METHOD GroupBuild : E_PROGRESS
VAR_INPUT
  Execute     : BOOL;
END_VAR
VAR_INST
  _nErrorId   : UDINT;
  _eJobReslt,
  _eState     : E_PROGRESS;
END_VAR
//-----------------------------------------------------------------------------
IF NOT Execute 
THEN 
	_eState                       := E_PROGRESS.PROGRESS_INIT; 
END_IF 
//-----------------------------------------------------------------------------
IF NOT Check() 
THEN 
	GroupBuild                    := E_PROGRESS.PROGRESS_ERROR; 
	RETURN; 
END_IF
//-----------------------------------------------------------------------------
//-----------------------------------------------------------------------------
CASE _eState
OF
  E_PROGRESS.PROGRESS_INIT:
    IF Execute
    THEN
      _nErrorId                 := 0;

      IF (_GroupInfo.AxisCount <> 0)
      THEN
        _nErrorId               := 9999;
        _eState                 := E_PROGRESS.PROGRESS_ERROR;
      ELSE
        _eState                 := E_PROGRESS.PROGRESS_BUSY;
        _eJobReslt              := _GroupItf.AddAll(FALSE);
      END_IF
    END_IF
END_CASE
//---------------------------------------------------------------------------
//---------------------------------------------------------------------------
CASE _eState
OF
  E_PROGRESS.PROGRESS_BUSY:
    _eJobReslt                  := _GroupItf.AddAll(TRUE);

    IF (_eJobReslt = E_PROGRESS.PROGRESS_ERROR)
    THEN
      _eState                   := E_PROGRESS.PROGRESS_ERROR;

      _nErrorId                 := _GroupInfo.GroupErrorId;
      _eJobReslt                := _GroupItf.AddAll(FALSE);

    ELSIF (_eJobReslt = E_PROGRESS.PROGRESS_DONE)
    THEN
      _eState                   := E_PROGRESS.PROGRESS_DONE;
      _eJobReslt                := _GroupItf.AddAll(FALSE);
    END_IF
END_CASE
//-----------------------------------------------------------------------------
//-----------------------------------------------------------------------------

GroupBuild                      := _eState;
END_METHOD

METHOD GroupClear : E_PROGRESS
VAR_INPUT
  Execute     : BOOL;
END_VAR
VAR_INST
  _nErrorId   : UDINT;
  _eJobReslt,
  _eState     : E_PROGRESS;
END_VAR
//-----------------------------------------------------------------------------
IF NOT Execute 
THEN 
	_eState                       := E_PROGRESS.PROGRESS_INIT; 
END_IF 
//-----------------------------------------------------------------------------
IF NOT Check() 
THEN 
	GroupClear                    := E_PROGRESS.PROGRESS_ERROR; 
	RETURN; 
END_IF
//-----------------------------------------------------------------------------
//-----------------------------------------------------------------------------
CASE _eState
OF
  E_PROGRESS.PROGRESS_INIT:
    IF Execute
    THEN
      _nErrorId                 := 0;
      _eJobReslt                := _GroupItf.McHaltAll(FALSE);
      _eState                   := E_PROGRESS.PROGRESS_BUSY;
    END_IF
  //---------------------------------------------------------------------------
  //---------------------------------------------------------------------------
  E_PROGRESS.PROGRESS_BUSY:
    _eJobReslt                  := _GroupItf.McHaltAll(TRUE);

    IF (_eJobReslt = E_PROGRESS.PROGRESS_ERROR)
    THEN
      _eState                   := E_PROGRESS.PROGRESS_ERROR;
      _nErrorId                 := _GroupInfo.GroupErrorId;
      _eJobReslt                := _GroupItf.McHaltAll(FALSE);

    ELSIF (_eJobReslt = E_PROGRESS.PROGRESS_DONE)
    THEN
      _eState                   := E_PROGRESS.PROGRESS_PREPARE;
      _eJobReslt                := _GroupItf.McResetAll(FALSE);
      _eJobReslt                := _GroupItf.McHaltAll(FALSE);
    END_IF
  //---------------------------------------------------------------------------
  //---------------------------------------------------------------------------
  E_PROGRESS.PROGRESS_PREPARE:
    _eJobReslt                  := _GroupItf.McResetAll(TRUE);

    IF (_eJobReslt = E_PROGRESS.PROGRESS_ERROR)
    THEN
      _eState                   := E_PROGRESS.PROGRESS_ERROR;
      _nErrorId                 := _GroupInfo.GroupErrorId;
      _eJobReslt                := _GroupItf.McResetAll(FALSE);

    ELSIF (_eJobReslt = E_PROGRESS.PROGRESS_DONE)
    THEN
      _eState                   := E_PROGRESS.PROGRESS_STARTUP;
      _eJobReslt                := _GroupItf.McResetAll(FALSE);
      _eJobReslt                := _GroupItf.RemoveAll(FALSE);
    END_IF
  //---------------------------------------------------------------------------
  //---------------------------------------------------------------------------
  E_PROGRESS.PROGRESS_STARTUP:
    _eJobReslt                  := _GroupItf.RemoveAll(TRUE);

    IF (_eJobReslt = E_PROGRESS.PROGRESS_ERROR)
    THEN
      _eState                   := E_PROGRESS.PROGRESS_ERROR;
      _nErrorId                 := _GroupInfo.GroupErrorId;
      _eJobReslt                := _GroupItf.RemoveAll(FALSE);

    ELSIF (_eJobReslt = E_PROGRESS.PROGRESS_DONE)
    THEN
      _eState                   := E_PROGRESS.PROGRESS_CHECK;
      _eJobReslt                := _GroupItf.RemoveAll(FALSE);
      _eJobReslt                := _GroupItf.Disable(FALSE);
    END_IF
  //---------------------------------------------------------------------------
  //---------------------------------------------------------------------------
  E_PROGRESS.PROGRESS_CHECK:
    _eJobReslt                  := _GroupItf.Disable(TRUE);

    IF (_eJobReslt = E_PROGRESS.PROGRESS_ERROR)
    THEN
      _eState                   := E_PROGRESS.PROGRESS_ERROR;
      _nErrorId                 := _GroupInfo.GroupErrorId;
      _eJobReslt                := _GroupItf.Disable(FALSE);

    ELSIF (_eJobReslt = E_PROGRESS.PROGRESS_DONE)
    THEN
      _eState                   := E_PROGRESS.PROGRESS_OCCUPIED;
      _eJobReslt                := _GroupItf.Disable(FALSE);
      _eJobReslt                := _GroupItf.Reset(FALSE);
    END_IF
  //---------------------------------------------------------------------------
  //---------------------------------------------------------------------------
  E_PROGRESS.PROGRESS_OCCUPIED:
    _eJobReslt                 := _GroupItf.Reset(TRUE);

    IF (_eJobReslt = E_PROGRESS.PROGRESS_ERROR)
    THEN
      _eState                   := E_PROGRESS.PROGRESS_ERROR;
      _nErrorId                 := _GroupInfo.GroupErrorId;
      _eJobReslt                := _GroupItf.Reset(FALSE);

    ELSIF (_eJobReslt = E_PROGRESS.PROGRESS_DONE)
    THEN
      _eState                   := E_PROGRESS.PROGRESS_WORKING;
      _eJobReslt                := _GroupItf.Reset(FALSE);
    END_IF
END_CASE
//-----------------------------------------------------------------------------
//-----------------------------------------------------------------------------
CASE _eState
OF
  E_PROGRESS.PROGRESS_WORKING:
    IF (_GroupInfo.GroupDisabled) AND NOT
       (_GroupInfo.GroupError)
    THEN
      _eState                   := E_PROGRESS.PROGRESS_DONE;
    ELSE
      IF (_GroupInfo.GroupErrorStop) OR
         (_GroupInfo.GroupError)
      THEN
        _eState                 := E_PROGRESS.PROGRESS_ERROR;
      END_IF
    END_IF
END_CASE
//-----------------------------------------------------------------------------
//-----------------------------------------------------------------------------

GroupClear                      := _eState;
END_METHOD

METHOD GroupEnable : E_PROGRESS
VAR_INPUT
  Execute     : BOOL;
END_VAR
VAR_INST
  _nErrorId   : UDINT;
  _eJobReslt,
  _eState     : E_PROGRESS;
END_VAR
//-----------------------------------------------------------------------------
IF NOT Execute 
THEN 
	_eState                       := E_PROGRESS.PROGRESS_INIT; 
END_IF 
//-----------------------------------------------------------------------------
IF NOT Check() 
THEN 
	GroupEnable                   := E_PROGRESS.PROGRESS_ERROR; 
	RETURN; 
END_IF
//-----------------------------------------------------------------------------
//-----------------------------------------------------------------------------
CASE _eState
OF
  E_PROGRESS.PROGRESS_INIT:
    IF Execute
    THEN
      _nErrorId                 := 0;

      IF NOT (_GroupInfo.AxisCount <> 0)
      THEN
        _nErrorId               := 9999;
        _eState                 := E_PROGRESS.PROGRESS_ERROR;
      ELSE
        _eState                 := E_PROGRESS.PROGRESS_BUSY;
        _eJobReslt              := _GroupItf.Enable(FALSE);
      END_IF
    END_IF
END_CASE
//---------------------------------------------------------------------------
//---------------------------------------------------------------------------
CASE _eState
OF
  E_PROGRESS.PROGRESS_BUSY:
    _eJobReslt                  := _GroupItf.Enable(TRUE);

    IF (_eJobReslt = E_PROGRESS.PROGRESS_ERROR)
    THEN
      _eState                   := E_PROGRESS.PROGRESS_ERROR;

      _nErrorId                 := _GroupInfo.GroupErrorId;
      _eJobReslt                := _GroupItf.Enable(FALSE);

    ELSIF (_eJobReslt = E_PROGRESS.PROGRESS_DONE)
    THEN
      _eState                   := E_PROGRESS.PROGRESS_CHECK;
      _eJobReslt                := _GroupItf.Enable(FALSE);
    END_IF
END_CASE
//-----------------------------------------------------------------------------
//-----------------------------------------------------------------------------
CASE _eState
OF
  E_PROGRESS.PROGRESS_CHECK:
    IF (_GroupInfo.GroupStandby) OR
       (_GroupInfo.GroupMoving)  OR
       (_GroupInfo.GroupNotReady)
    THEN
      _eState                   := E_PROGRESS.PROGRESS_DONE;
    ELSE
      IF (_GroupInfo.GroupErrorStop) OR
         (_GroupInfo.GroupError)
      THEN
        _eState                 := E_PROGRESS.PROGRESS_ERROR;
      END_IF
    END_IF
END_CASE
//-----------------------------------------------------------------------------
//-----------------------------------------------------------------------------
GroupEnable                     := _eState;
END_METHOD

PROPERTY GroupInfo : REFERENCE TO ST_GROUP_INFO
SET
_GroupInfo REF= GroupInfo;
END_SET
END_PROPERTY

PROPERTY GroupItf : I_XtsTransport_CaGroup
SET
_GroupItf := GroupItf;
END_SET
END_PROPERTY

METHOD MoverDisableAll : e_progress
VAR_INPUT
  Execute     : BOOL;
END_VAR
VAR_INST
  _nMover     : UINT;
  _nErrorId   : UDINT;
  _eRslt,
  _eState     : E_PROGRESS;
END_VAR
//-----------------------------------------------------------------------------
IF NOT Execute 
THEN 
	_eState                       := E_PROGRESS.PROGRESS_INIT; 
END_IF 
//-----------------------------------------------------------------------------
IF NOT Check() 
THEN 
	MoverDisableAll               := E_PROGRESS.PROGRESS_ERROR; 
	RETURN; 
END_IF
//-----------------------------------------------------------------------------
//-----------------------------------------------------------------------------
CASE _eState
OF
  E_PROGRESS.PROGRESS_INIT:
    IF Execute
    THEN
      _nErrorId                 := 0;
      _nMover                   := 1;

      _eState                   := E_PROGRESS.PROGRESS_BUSY;
    END_IF
END_CASE
//-----------------------------------------------------------------------------
//-----------------------------------------------------------------------------
CASE _eState
OF
  E_PROGRESS.PROGRESS_BUSY:
    _eState                     := E_PROGRESS.PROGRESS_PREPARE;
    _eRslt                      := _MoverItf[_nMover].Disable(FALSE);
END_CASE
//-----------------------------------------------------------------------------
//-----------------------------------------------------------------------------
CASE _eState
OF
  E_PROGRESS.PROGRESS_PREPARE:
    _eRslt                      := _MoverItf[_nMover].Disable(TRUE);

    IF (_eRslt = E_PROGRESS.PROGRESS_ERROR)
    THEN
      _eState                   := E_PROGRESS.PROGRESS_ERROR;
      _nErrorId                 := _MoverInfo[_nMover].nErrorId; 

    ELSIF (_eRslt = E_PROGRESS.PROGRESS_DONE)
    THEN
      _eState                   := E_PROGRESS.PROGRESS_STARTUP;
    END_IF
END_CASE
//-----------------------------------------------------------------------------
//-----------------------------------------------------------------------------
CASE _eState
OF
  E_PROGRESS.PROGRESS_STARTUP:
    _eState                     := E_PROGRESS.PROGRESS_CHECK;
    _eRslt                      := _MoverItf[_nMover].Disable(FALSE);
END_CASE
//-----------------------------------------------------------------------------
//-----------------------------------------------------------------------------
CASE _eState
OF
  E_PROGRESS.PROGRESS_CHECK:
    IF (_nMover > MAX_MOVER-1)
    THEN
      _eState                   := E_PROGRESS.PROGRESS_DONE;
    ELSE
      _nMover                   := _nMover + 1;
      _eState                   := E_PROGRESS.PROGRESS_BUSY;
    END_IF
END_CASE
//-----------------------------------------------------------------------------
//-----------------------------------------------------------------------------

MoverDisableAll                 := _eState;
END_METHOD

METHOD MoverEnableAll : e_progress
VAR_INPUT
  Execute     : BOOL;
END_VAR
VAR_INST
  _nMover     : UINT;
  _nErrorId   : UDINT;
  _eRslt,
  _eState     : E_PROGRESS;
END_VAR
//-----------------------------------------------------------------------------
IF NOT Execute 
THEN 
	_eState                       := E_PROGRESS.PROGRESS_INIT; 
END_IF 
//-----------------------------------------------------------------------------
IF NOT Check() 
THEN 
	MoverEnableAll                := E_PROGRESS.PROGRESS_ERROR; 
	RETURN; 
END_IF
//-----------------------------------------------------------------------------
//-----------------------------------------------------------------------------
CASE _eState
OF
  E_PROGRESS.PROGRESS_INIT:
    IF Execute
    THEN
      _nErrorId                 := 0;
      _nMover                   := 1;

      _eState                   := E_PROGRESS.PROGRESS_BUSY;
    END_IF
END_CASE
//-----------------------------------------------------------------------------
//-----------------------------------------------------------------------------
CASE _eState
OF
  E_PROGRESS.PROGRESS_BUSY:
    _eState                     := E_PROGRESS.PROGRESS_PREPARE;
    _eRslt                      := _MoverItf[_nMover].Enable(FALSE);
END_CASE
//-----------------------------------------------------------------------------
//-----------------------------------------------------------------------------
CASE _eState
OF
  E_PROGRESS.PROGRESS_PREPARE:
    _eRslt                      := _MoverItf[_nMover].Enable(TRUE);

    IF (_eRslt = E_PROGRESS.PROGRESS_ERROR)
    THEN
      _eState                   := E_PROGRESS.PROGRESS_ERROR;
      _nErrorId                 := _MoverInfo[_nMover].nErrorId; 

    ELSIF (_eRslt = E_PROGRESS.PROGRESS_DONE)
    THEN
      _eState                   := E_PROGRESS.PROGRESS_STARTUP;
    END_IF
END_CASE
//-----------------------------------------------------------------------------
//-----------------------------------------------------------------------------
CASE _eState
OF
  E_PROGRESS.PROGRESS_STARTUP:
    _eState                     := E_PROGRESS.PROGRESS_CHECK;
    _eRslt                      := _MoverItf[_nMover].Enable(FALSE);
END_CASE
//-----------------------------------------------------------------------------
//-----------------------------------------------------------------------------
CASE _eState
OF
  E_PROGRESS.PROGRESS_CHECK:
    IF (_nMover > MAX_MOVER-1)
    THEN
      _eState                   := E_PROGRESS.PROGRESS_DONE;
    ELSE
      _nMover                   := _nMover + 1;
      _eState                   := E_PROGRESS.PROGRESS_BUSY;
    END_IF
END_CASE
//-----------------------------------------------------------------------------
//-----------------------------------------------------------------------------

MoverEnableAll                  := _eState;
END_METHOD

PROPERTY MoverInfo : REFERENCE TO ARRAY[1..MAX_MOVER] OF ST_MOVER_INFO
SET
_MoverInfo REF= MoverInfo;
END_SET
END_PROPERTY

PROPERTY MoverItf : reference TO ARRAY[1..MAX_MOVER] OF I_XtsTransport_Mover
SET
_MoverItf REF= MoverItf;
END_SET
END_PROPERTY

PROPERTY StartStationIndex : uint
GET
StartStationIndex := _nStartStation;
END_GET
SET
_nStartStation := StartStationIndex;
END_SET
END_PROPERTY

PROPERTY State : REFERENCE TO ST_XTS_TRANSPORT_STATE
SET
_State ref= State;
END_SET
END_PROPERTY

PROPERTY StationCtrlItf : REFERENCE TO ARRAY[1..MAX_STATION]  OF I_XtsTransport_Station;
SET
_ItfStationCtrl REF= StationCtrlItf;
END_SET
END_PROPERTY

PROPERTY StationListsItf : reference to ARRAY[1..MAX_STATION] OF I_Station_LinkedList
SET
_ItfStationList ref= StationListsItf;
END_SET
END_PROPERTY

PROPERTY StationStart : reference to ST_STATION_PARAMETER
SET
_StationStart REF= StationStart;
END_SET
END_PROPERTY

METHOD Template : E_PROGRESS
VAR_INPUT
  Execute     : BOOL;
END_VAR
VAR_INST
  _nErrorId   : UDINT;
  _eState     : E_PROGRESS;
END_VAR
//-----------------------------------------------------------------------------
IF NOT Execute 
THEN 
	_eState                       := E_PROGRESS.PROGRESS_INIT; 
END_IF 
//-----------------------------------------------------------------------------
IF NOT Check() 
THEN 
	Template_1                    := E_PROGRESS.PROGRESS_ERROR; 
	RETURN; 
END_IF
//-----------------------------------------------------------------------------
//-----------------------------------------------------------------------------
CASE _eState
OF
  E_PROGRESS.PROGRESS_INIT:
    IF Execute
    THEN
      _nErrorId                 := 0;

      _eState                   := E_PROGRESS.PROGRESS_BUSY;
    END_IF
END_CASE
//-----------------------------------------------------------------------------
//-----------------------------------------------------------------------------
CASE _eState
OF
  E_PROGRESS.PROGRESS_BUSY:
    _eState                     := E_PROGRESS.PROGRESS_PREPARE;
END_CASE
//-----------------------------------------------------------------------------
//-----------------------------------------------------------------------------
CASE _eState
OF
  E_PROGRESS.PROGRESS_PREPARE:

    IF (.Error)
    THEN
      _eState                   := E_PROGRESS.PROGRESS_ERROR;
      _nErrorId                 := 


    ELSIF (.Done)
    THEN
      _eState                   := E_PROGRESS.;

    END_IF
END_CASE
//-----------------------------------------------------------------------------
//-----------------------------------------------------------------------------

Template_1                      := _eState;
END_METHOD

METHOD TransportRestart : e_progress
VAR_INPUT
  Execute     : BOOL;
END_VAR
VAR_INST
  _nMover     : UINT;
  _nErrorId   : UDINT;
  _eRslt,
  _eState     : E_PROGRESS;
END_VAR
//-----------------------------------------------------------------------------
IF NOT Execute 
THEN 
	_eState                       := E_PROGRESS.PROGRESS_INIT; 
END_IF 
//-----------------------------------------------------------------------------
IF NOT Check() 
THEN 
	TransportRestart              := E_PROGRESS.PROGRESS_ERROR; 
	RETURN; 
END_IF
//-----------------------------------------------------------------------------
//-----------------------------------------------------------------------------
CASE _eState
OF
  E_PROGRESS.PROGRESS_INIT:
    IF Execute
    THEN
      _nErrorId                 := 0;
      _nMover                   := 1;

      _eState                   := E_PROGRESS.PROGRESS_BUSY;
    END_IF
END_CASE
//-----------------------------------------------------------------------------
//-----------------------------------------------------------------------------
CASE _eState
OF
  E_PROGRESS.PROGRESS_BUSY:
    _eState                     := E_PROGRESS.PROGRESS_PREPARE;

END_CASE
//-----------------------------------------------------------------------------
//-----------------------------------------------------------------------------
CASE _eState
OF
  E_PROGRESS.PROGRESS_PREPARE:


    IF (_eRslt = E_PROGRESS.PROGRESS_ERROR)
    THEN
      _eState                   := E_PROGRESS.PROGRESS_ERROR;
      _nErrorId                 := _MoverInfo[_nMover].nErrorId; 

    ELSIF (_eRslt = E_PROGRESS.PROGRESS_DONE)
    THEN
      _eState                   := E_PROGRESS.PROGRESS_STARTUP;
    END_IF
END_CASE
//-----------------------------------------------------------------------------
//-----------------------------------------------------------------------------
CASE _eState
OF
  E_PROGRESS.PROGRESS_STARTUP:
    _eState                     := E_PROGRESS.PROGRESS_CHECK;

END_CASE
//-----------------------------------------------------------------------------
//-----------------------------------------------------------------------------
CASE _eState
OF
  E_PROGRESS.PROGRESS_CHECK:
    IF (_nMover > MAX_MOVER-1)
    THEN
      _eState                   := E_PROGRESS.PROGRESS_DONE;
    ELSE
      _nMover                   := _nMover + 1;
      _eState                   := E_PROGRESS.PROGRESS_BUSY;
    END_IF
END_CASE
//-----------------------------------------------------------------------------
//-----------------------------------------------------------------------------

TransportRestart                := _eState;
END_METHOD

METHOD TransportStart : e_progress
VAR_INPUT
  Execute       : BOOL;
END_VAR
VAR_INST
  _nMover,
  _nStation     : UINT;
  _nErrorId     : UDINT;

  _stMoveData   : ST_MOVE_DATA;

  _eRslt,
  _eState       : E_PROGRESS;

END_VAR
//-----------------------------------------------------------------------------
IF NOT Execute 
THEN 
	_eState                       := E_PROGRESS.PROGRESS_INIT; 
END_IF 
//-----------------------------------------------------------------------------
IF NOT Check() 
THEN 
	TransportStart                := E_PROGRESS.PROGRESS_ERROR; 
	RETURN; 
END_IF
//-----------------------------------------------------------------------------
//-----------------------------------------------------------------------------
CASE _eState
OF
  E_PROGRESS.PROGRESS_INIT:
    IF Execute
    THEN
      _nErrorId                 := 0;
      _nMover                   := 1;

      IF (_StationStart.rPosWait - _MoverInfo[_nMover].rModuloActPos < 0)
      THEN
        _stMoveData.rPos        := _StationStart.rPosWait + _MoverItf[_nMover].RailLength;
      ELSE
        _stMoveData.rPos        := _StationStart.rPosWait;
      END_IF

      _stMoveData.rGap          := _StationStart.rGap;

      _stMoveData.rVelo         := _StationStart.rVelo;
      _stMoveData.rAcc          := _StationStart.rAccDec;
      _stMoveData.rJerk         := _StationStart.rJerk;

      _stMoveData.rDelta        :=   0.05;
      _stMoveData.rDistance     :=  -1.0;     // distance used by SendToPosCa

      _stMoveData.rOverride     := 100.0;

      FOR _nStation := 1 TO MAX_STATION
      DO
        _ItfStationCtrl[_nStation].Init();    // clear all stations
      END_FOR

      _eState                   := E_PROGRESS.PROGRESS_BUSY;
    END_IF

  //---------------------------------------------------------------------------
  E_PROGRESS.PROGRESS_BUSY:
    _eState                     := E_PROGRESS.PROGRESS_PREPARE;
    _eRslt                      := _MoverItf[_nMover].SendToModuloPosCa(FALSE, _stMoveData);
    _eRslt                      := _MoverItf[_nMover].SendToAbsPosCa(FALSE, _stMoveData);

  E_PROGRESS.PROGRESS_PREPARE:
    _eRslt                      := _MoverItf[_nMover].SendToModuloPosCa(TRUE, _stMoveData);

    IF (_eRslt = E_PROGRESS.PROGRESS_ERROR)
    THEN
      _eState                   := E_PROGRESS.PROGRESS_ERROR;
      _nErrorId                 := _MoverInfo[_nMover].nErrorId;
      _eRslt                    := _MoverItf[_nMover].SendToModuloPosCa(FALSE, _stMoveData); 

    ELSIF (_eRslt = E_PROGRESS.PROGRESS_DONE)
    THEN
      _eState                   := E_PROGRESS.PROGRESS_STARTUP;
      _eRslt                    := _MoverItf[_nMover].SendToModuloPosCa(FALSE, _stMoveData);
    END_IF

  //---------------------------------------------------------------------------
  E_PROGRESS.PROGRESS_STARTUP:
    IF (_nMover > MAX_MOVER-1)
    THEN
      // all mover are sent to start position, now prepare ticket for Mover 1
      _eState                         := E_PROGRESS.PROGRESS_CHECK;
      // ticket data
      _stMoverDataSend.nMask          := TO_USINT(EXPT(2,_StationStart.nConfiguredStopCount))-1;
      _stMoverDataSend.nMoverId       := TO_USINT(1);
      _stMoverDataSend.nTargetStation := TO_USINT(_nStartStation);
  
      _stListResult                   := _ItfStationList[_nStartStation].AddTailValue(_stMoverDataSend); // add first mover to list of _ItfStations[_nStartStation]

    ELSE
      _nMover                   := _nMover + 1;                                                 // increment mover ID
      _stMoveData.rPos          := _StationStart.rPosWait + 2*_MoverItf[_nMover].RailLength;    // all other mover are commanded an extra round, to make sure that mover 1 is always leading the pack
      _eState                   := E_PROGRESS.PROGRESS_BUSY;                                    // go back and trigger move
    END_IF

  //---------------------------------------------------------------------------
  E_PROGRESS.PROGRESS_CHECK:
    IF (_MoverInfo[1].rAbsActPos > _MoverInfo[1].rAbsTargetPos - 1.0) AND
       (_MoverInfo[1].rAbsActPos < _MoverInfo[1].rAbsTargetPos + 1.0) // wait for first mover to arrive
    THEN
      IF (_GroupInfo.AllAxesStanding) // wait for all mover standstill
      THEN
        _stMoveData.rPos        := _MoverInfo[1].rAbsTargetPos;                    // Mover1 position to retrigger the movers

        IF (MAX_MOVER > 1)
        THEN
          _nMover               := 2;
          IF (_stMoveData.rPos < _MoverInfo[_nMover].rAbsActPos)
          THEN
            _stMoveData.rPos    := _stMoveData.rPos + _MoverItf[_nMover].RailLength;
          END_IF
          _eState               := E_PROGRESS.PROGRESS_OCCUPIED;
        ELSE
          _eState               := E_PROGRESS.PROGRESS_WORKING;
        END_IF
      END_IF
    END_IF

  //---------------------------------------------------------------------------
  E_PROGRESS.PROGRESS_OCCUPIED:
    _eRslt                      := _MoverItf[_nMover].SendToAbsPosCa(TRUE, _stMoveData); // retrigger

    IF (_eRslt = E_PROGRESS.PROGRESS_ERROR)
    THEN
      _eState                   := E_PROGRESS.PROGRESS_ERROR;
      _nErrorId                 := _MoverInfo[_nMover].nErrorId;
      _eRslt                    := _MoverItf[_nMover].SendToAbsPosCa(FALSE, _stMoveData); 

    ELSIF (_eRslt = E_PROGRESS.PROGRESS_DONE)
    THEN
      _eState                   := E_PROGRESS.PROGRESS_WORKING;
      _eRslt                    := _MoverItf[_nMover].SendToAbsPosCa(FALSE, _stMoveData);

      // write ticket for mover in station list
      _stMoverDataSend.nMask          := TO_USINT(EXPT(2,_StationStart.nConfiguredStopCount))-1;
      _stMoverDataSend.nMoverId       := TO_USINT(_nMover);
      _stMoverDataSend.nTargetStation := TO_USINT(_nStartStation);
  
      _stListResult                   := _ItfStationList[_nStartStation].AddTailValue(_stMoverDataSend); // enter in list
    END_IF

  //---------------------------------------------------------------------------
  E_PROGRESS.PROGRESS_WORKING:
    IF (_nMover > MAX_MOVER-1)
    THEN
      _eState                   := E_PROGRESS.PROGRESS_DONE;
    ELSE
      _nMover                   := _nMover + 1;
      IF (_stMoveData.rPos < _MoverInfo[_nMover].rAbsActPos)
      THEN
        _stMoveData.rPos        := _stMoveData.rPos + _MoverItf[_nMover].RailLength;
      END_IF
      _eState                   := E_PROGRESS.PROGRESS_OCCUPIED;
    END_IF
END_CASE
//-----------------------------------------------------------------------------
//-----------------------------------------------------------------------------

TransportStart                  := _eState;
END_METHOD

PROPERTY XpuCtrl : REFERENCE TO ST_XPU_CTRL
SET
_XpuCtrl REF= XpuCtrl;
END_SET
END_PROPERTY

PROPERTY XpuInfo : REFERENCE TO ST_XPU_INFO
SET
_XpuInfo REF= XpuInfo;
END_SET
END_PROPERTY

METHOD XpuInit : E_PROGRESS
VAR_INPUT
  Execute     : BOOL;
END_VAR
VAR_INST
  _nErrorId   : UDINT;
  _eJobReslt,
  _eState     : E_PROGRESS;
END_VAR
//-----------------------------------------------------------------------------
IF NOT Execute 
THEN 
	_eState                       := E_PROGRESS.PROGRESS_INIT; 
END_IF 
//-----------------------------------------------------------------------------
IF NOT Check() 
THEN 
	XpuInit                       := E_PROGRESS.PROGRESS_ERROR; 
	RETURN; 
END_IF
//-----------------------------------------------------------------------------
//-----------------------------------------------------------------------------
CASE _eState
OF
  E_PROGRESS.PROGRESS_INIT:
    IF Execute
    THEN
      _nErrorId                 := 0;
      _XpuCtrl.Cmd              := E_XPU_CTRL.XTS_CMD_NULL; // clear interface

      _eState                   := E_PROGRESS.PROGRESS_BUSY;
    END_IF
  //---------------------------------------------------------------------------
  //---------------------------------------------------------------------------
  E_PROGRESS.PROGRESS_BUSY:
    _XpuCtrl.Cmd                := E_XPU_CTRL.XTS_CMD_INIT; // start Xpu init

    IF (f_GetProgress(_XpuState.State) = E_PROGRESS.PROGRESS_DONE)         // check Xpu init done
    THEN
      _eState                   := E_PROGRESS.PROGRESS_PREPARE;

    ELSIF (f_GetProgress(_XpuState.State) = E_PROGRESS.PROGRESS_ERROR)     // check for error
    THEN
      _eState                   := E_PROGRESS.PROGRESS_ERROR;
    END_IF
  //---------------------------------------------------------------------------
  //---------------------------------------------------------------------------
  E_PROGRESS.PROGRESS_PREPARE:
    _XpuCtrl.Cmd                := E_XPU_CTRL.XTS_IDLE;     // Xpu start cyclic checks and mover detection

    IF (f_GetProgress(_XpuState.State) = E_PROGRESS.PROGRESS_ERROR)     // check for error
    THEN
      _eState                   := E_PROGRESS.PROGRESS_ERROR;

    ELSIF (f_GetProgress(_XpuState.State) = E_PROGRESS.PROGRESS_WORKING)      // check Xpu Idle working
    THEN
      _eState                   := E_PROGRESS.PROGRESS_STARTUP;

    END_IF
  //---------------------------------------------------------------------------
  //---------------------------------------------------------------------------
  E_PROGRESS.PROGRESS_STARTUP:
    IF (f_GetProgress(_XpuState.State) = E_PROGRESS.PROGRESS_ERROR)
    THEN
      _eState                   := E_PROGRESS.PROGRESS_ERROR;

    ELSIF (_XpuState.Check = E_XPU_CHECK.MOVER_ID_SIMULATION) OR
          (_XpuState.Check = E_XPU_CHECK.MOVER_ID_STANDARD)   OR
          (_XpuState.Check = E_XPU_CHECK.MOVER_ID_DETECTION_VALID)
    THEN
      _eState                   := E_PROGRESS.PROGRESS_DONE;
    END_IF
END_CASE
//-----------------------------------------------------------------------------
//-----------------------------------------------------------------------------
XpuInit                         := _eState;
END_METHOD

PROPERTY XpuState : REFERENCE TO ST_XPU_STATE
SET
_XpuState ref= XpuState;
END_SET
END_PROPERTY

END_FUNCTION_BLOCK

// ---- GlobalTextList.TcGTLO
TEXTLIST GlobalTextList
  17 = ' STATION_ENABLE'
  34 = ' STATION_MOVER_ENTER'
  452 = ' STATION_MOVER_GONE'
  75 = ' STATION_MOVER_OUT'
  598 = ' STATION_PROCESS_DONE'
  750 = ' STATION_PROCESS_START'
  294 = '%.2f'
  191 = '%d'
  836 = '%s'
  563 = '.nMask'
  249 = '.nMoverId'
  822 = '.nTargetStation'
  663 = '.rOffset'
  248 = 'Activate'
  444 = 'Activate Visu list'
  704 = 'All Positions Valid'
  562 = 'AllAxisStanding'
  878 = 'AxisCount Enabled: %d'
  162 = 'AxisCount: %d'
  914 = 'ConstantVelocity'
  929 = 'Control'
  707 = 'CyclicCheck: %s'
  660 = 'DC Link All Modules'
  359 = 'Decelerating'
  843 = 'Detected AxisCount: %d'
  243 = 'eDevice'
  244 = 'eSubdevice'
  242 = 'eType'
  772 = 'Expected AxisCount: %d'
  48 = 'GroupDisabled'
  915 = 'GroupError'
  495 = 'GroupErrorId: %d'
  975 = 'GroupErrorStop'
  940 = 'GroupHoming'
  300 = 'GroupMoving'
  807 = 'GroupNotReady'
  438 = 'GroupStandby'
  226 = 'GroupStatusBusy'
  204 = 'GroupStatusValid'
  973 = 'GroupStopping'
  942 = 'GVL_XTS.CaGroupInfo'
  680 = 'ID Detection Active'
  238 = 'ID Detection Error'
  526 = 'ID Detection Mode: %s'
  29 = 'ID Detection Valid'
  245 = 'iErrorNumber'
  211 = 'Info Act Pos Absolute'
  586 = 'Info Act Pos Modulo'
  21 = 'Info Mover Avoiding Collision'
  282 = 'Info Mover Coupled'
  398 = 'Info Mover Enabled'
  751 = 'Info Mover Error'
  907 = 'Info Mover Standstill'
  480 = 'Info nError ID'
  922 = 'Info Target Pos Absolute'
  16 = 'Info Target Pos Modulo'
  616 = 'InPosition'
  713 = 'Mask: %b'
  972 = 'Mask: %d'
  779 = 'Mask: %s'
  726 = 'McGroupState:      %s'
  160 = 'McGroupState: %d  %s'
  974 = 'MOVER command'
  387 = 'Mover ID: %d'
  297 = 'Mover Position Assignement: %s'
  840 = 'MOVER result:  %s'
  53 = 'MOVER state:   %s'
  756 = 'nMoverSelected: %d'
  669 = 'nStation selected: %d'
  94 = 'Offset %.3f'
  427 = 'Offset: %.3f'
  312 = 'Operation Mode: %s'
  320 = 'Queue: %d'
  91 = 'Set Acceleration'
  399 = 'Set Delta'
  382 = 'Set Distance'
  757 = 'Set Gap'
  934 = 'Set Jerk'
  201 = 'Set Override'
  936 = 'Set Position'
  62 = 'Set Velocity'
  231 = 'State'
  748 = 'Station Control'
  267 = 'Station State'
  627 = 'STATION_ENABLE'
  247 = 'sText'
  54 = 'Target Station %d'
  567 = 'Target Station: %d'
  246 = 'tTime'
  517 = 'WRITE TO FILE'
  275 = 'XPU Command'
  227 = 'XpuResult:   %s'
  96 = 'XpuState:    %s'
  884 = 'XTS Station'
  572 = 'XTS Transport Check:  %s'
  212 = 'XTS Transport Check: %s'
  500 = 'XTS Transport Command'
  395 = 'XTS Transport Result: %s'
  798 = 'XTS Transport State:  %s'
  417 = 'XTS Transport State: %s'
END_TEXTLIST

// ---- XTS/_Visualization/GROUP_VISU.TcVIS
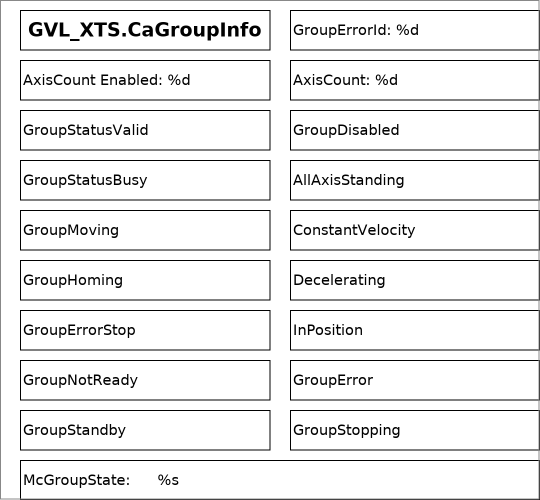
VISUALIZATION GROUP_VISU  // 540x500
    Rectangle (20,110 250x40), "GroupStatusValid", colour toggle: GVL_XTS.XtsTransportState.GroupInfo.GroupStatusValid
    Rectangle (20,160 250x40), "GroupStatusBusy", colour toggle: GVL_XTS.XtsTransportState.GroupInfo.GroupStatusBusy
    Rectangle (20,210 250x40), "GroupMoving", colour toggle: GVL_XTS.XtsTransportState.GroupInfo.GroupMoving
    Rectangle (20,260 250x40), "GroupHoming", colour toggle: GVL_XTS.XtsTransportState.GroupInfo.GroupHoming
    Rectangle (20,310 250x40), "GroupErrorStop", colour toggle: GVL_XTS.XtsTransportState.GroupInfo.GroupErrorStop
    Rectangle (20,360 250x40), "GroupNotReady", colour toggle: GVL_XTS.XtsTransportState.GroupInfo.GroupNotReady
    Rectangle (20,410 250x40), "GroupStandby", colour toggle: GVL_XTS.XtsTransportState.GroupInfo.GroupStandby
    Rectangle (290,410 250x40), "GroupStopping", colour toggle: GVL_XTS.XtsTransportState.GroupInfo.GroupStopping
    Rectangle (290,110 250x40), "GroupDisabled", colour toggle: GVL_XTS.XtsTransportState.GroupInfo.GroupDisabled
    Rectangle (290,160 250x40), "AllAxisStanding", colour toggle: GVL_XTS.XtsTransportState.GroupInfo.AllAxesStanding
    Rectangle (290,210 250x40), "ConstantVelocity", colour toggle: GVL_XTS.XtsTransportState.GroupInfo.ConstantVelocity
    Rectangle (290,260 250x40), "Decelerating", colour toggle: GVL_XTS.XtsTransportState.GroupInfo.Decelerating
    Rectangle (290,310 250x40), "InPosition", colour toggle: GVL_XTS.XtsTransportState.GroupInfo.InPosition
    Rectangle (290,360 250x40), "GroupError", colour toggle: GVL_XTS.XtsTransportState.GroupInfo.GroupError
    Rectangle (290,10 250x40), "GroupErrorId: %d", text variable: GVL_XTS.XtsTransportState.GroupInfo.GroupErrorId
    Rectangle (290,60 250x40), "AxisCount: %d", text variable: GVL_XTS.XtsTransportState.GroupInfo.AxisCount
    Rectangle (20,460 520x40), "McGroupState: %s", text variable: MAIN.sCaGroupState
    Rectangle (20,10 250x40), "GVL_XTS.CaGroupInfo"
    Rectangle (20,60 250x40), "AxisCount Enabled: %d", text variable: GVL_XTS.CaGroupInfo.AxisCountEnabled
END_VISUALIZATION
